PROGRAM MAIN
VAR
END_VAR

END_PROGRAM

(* stored: Version 1.1.0.1
   POU MAIN: Id {31fc8197-d1d1-4826-96a3-9abbcc26a250} *)
